LIN {X 0,Y 45.733,Z 728.488,A -85,B 0,C 180,E1 -30032.551,E2 -30032.551} C_VEL
LIN {X 0,Y 45.215,Z 723.563,A -85,B 0,C 180,E1 -30078.116,E2 -30078.116} C_VEL
LIN {X 0,Y 55.921,Z 720.857,A -85,B 0,C 180,E1 -30098.935,E2 -30098.935} C_VEL
LIN {X 0,Y 58.826,Z 720.679,A -85,B 0,C 180,E1 -30104.197,E2 -30104.197} C_VEL
LIN {X 0,Y 48.539,Z 726.04,A -85,B 0,C 180,E1 -30114.598,E2 -30114.598} C_VEL
LIN {X 0,Y 40.212,Z 730.336,A -85,B 0,C 180,E1 -30129.529,E2 -30129.529} C_VEL
LIN {X 0,Y 35.144,Z 733.679,A -85,B 0,C 180,E1 -30150.436,E2 -30150.436} C_VEL
LIN {X 0,Y 34.555,Z 735.898,A -85,B 0,C 180,E1 -30173.989,E2 -30173.989} C_VEL
LIN {X 0,Y 39.075,Z 737.272,A -85,B 0,C 180,E1 -30195.991,E2 -30195.991} C_VEL
LIN {X 0,Y 49.391,Z 737.543,A -85,B 0,C 180,E1 -30214.726,E2 -30214.726} C_VEL
LIN {X 0,Y 63.722,Z 736.291,A -85,B 0,C 180,E1 -30227.254,E2 -30227.254} C_VEL
LIN {X 0,Y 79.407,Z 733.489,A -85,B 0,C 180,E1 -30234.92,E2 -30234.92} C_VEL
LIN {X 0,Y 80.609,Z 733.2,A -85,B 0,C 180,E1 -30235.369,E2 -30235.369} C_VEL
LIN {X 0,Y 83.762,Z 732.473,A -85,B 0,C 180,E1 -30236.987,E2 -30236.987} C_VEL
LIN {X 0,Y 92.73,Z 730.259,A -85,B 0,C 180,E1 -30243.394,E2 -30243.394} C_VEL
LIN {X 0,Y 96.102,Z 729.265,A -85,B 0,C 180,E1 -30244.536,E2 -30244.536} C_VEL
LIN {X 0,Y 98.768,Z 728.439,A -85,B 0,C 180,E1 -30245.06,E2 -30245.06} C_VEL
LIN {X 0,Y 98.879,Z 728.459,A -85,B 0,C 180,E1 -30245.741,E2 -30245.741} C_VEL
LIN {X 0,Y 85.239,Z 732.788,A -85,B 0,C 180,E1 -30248.386,E2 -30248.386} C_VEL
LIN {X 0,Y 71.87,Z 736.158,A -85,B 0,C 180,E1 -30252.108,E2 -30252.108} C_VEL
LIN {X 0,Y 58.961,Z 738.548,A -85,B 0,C 180,E1 -30257.552,E2 -30257.552} C_VEL
LIN {X 0,Y 44.77,Z 740.255,A -85,B 0,C 180,E1 -30268.091,E2 -30268.091} C_VEL
LIN {X 0,Y 32.272,Z 740.603,A -85,B 0,C 180,E1 -30289.225,E2 -30289.225} C_VEL
LIN {X 0,Y 27.769,Z 739.764,A -85,B 0,C 180,E1 -30315.356,E2 -30315.356} C_VEL
LIN {X 0,Y 27.901,Z 739.026,A -85,B 0,C 180,E1 -30330.015,E2 -30330.015} C_VEL
LIN {X 0,Y 29.362,Z 736.41,A -85,B 0,C 180,E1 -30358.618,E2 -30358.618} C_VEL
LIN {X 0,Y 36.467,Z 732.693,A -85,B 0,C 180,E1 -30380.451,E2 -30380.451} C_VEL
LIN {X 0,Y 39.799,Z 730.817,A -85,B 0,C 180,E1 -30388.016,E2 -30388.016} C_VEL
LIN {X 0,Y 38.938,Z 726.095,A -85,B 0,C 180,E1 -30441.165,E2 -30441.165} C_VEL
LIN {X 0,Y 48.749,Z 723.861,A -85,B 0,C 180,E1 -30460.968,E2 -30460.968} C_VEL
LIN {X 0,Y 48.378,Z 724.351,A -85,B 0,C 180,E1 -30463.406,E2 -30463.406} C_VEL
LIN {X 0,Y 37.896,Z 729.071,A -85,B 0,C 180,E1 -30476.182,E2 -30476.182} C_VEL
LIN {X 0,Y 30.159,Z 732.784,A -85,B 0,C 180,E1 -30496.51,E2 -30496.51} C_VEL
LIN {X 0,Y 27.913,Z 734.288,A -85,B 0,C 180,E1 -30509.985,E2 -30509.985} C_VEL
LIN {X 0,Y 27.959,Z 736.485,A -85,B 0,C 180,E1 -30540.163,E2 -30540.163} C_VEL
LIN {X 0,Y 34.279,Z 737.777,A -85,B 0,C 180,E1 -30565.072,E2 -30565.072} C_VEL
LIN {X 0,Y 45.412,Z 738.013,A -85,B 0,C 180,E1 -30581.965,E2 -30581.965} C_VEL
LIN {X 0,Y 61.119,Z 736.803,A -85,B 0,C 180,E1 -30593.394,E2 -30593.394} C_VEL
LIN {X 0,Y 70.34,Z 735.461,A -85,B 0,C 180,E1 -30597.481,E2 -30597.481} C_VEL
LIN {X 0,Y 84.374,Z 732.503,A -85,B 0,C 180,E1 -30601.894,E2 -30601.894} C_VEL
LIN {X 0,Y 96.102,Z 729.265,A -85,B 0,C 180,E1 -30604.536,E2 -30604.536} C_VEL
LIN {X 0,Y 95.247,Z 729.582,A -85,B 0,C 180,E1 -30604.95,E2 -30604.95} C_VEL
LIN {X 0,Y 89.533,Z 731.374,A -85,B 0,C 180,E1 -30605.285,E2 -30605.285} C_VEL
LIN {X 0,Y 76.501,Z 734.548,A -85,B 0,C 180,E1 -30604.408,E2 -30604.408} C_VEL
LIN {X 0,Y 67.963,Z 736.139,A -85,B 0,C 180,E1 -30602.933,E2 -30602.933} C_VEL
LIN {X 0,Y 65.186,Z 736.543,A -85,B 0,C 180,E1 -30602.135,E2 -30602.135} C_VEL
LIN {X 0,Y 49.356,Z 738.175,A -85,B 0,C 180,E1 -30595.276,E2 -30595.276} C_VEL
LIN {X 0,Y 36.402,Z 738.534,A -85,B 0,C 180,E1 -30584.821,E2 -30584.821} C_VEL
LIN {X 0,Y 25.651,Z 737.78,A -85,B 0,C 180,E1 -30565.251,E2 -30565.251} C_VEL
LIN {X 0,Y 20.031,Z 736.132,A -85,B 0,C 180,E1 -30530.517,E2 -30530.517} C_VEL
LIN {X 0,Y 21.174,Z 734.546,A -85,B 0,C 180,E1 -30504.822,E2 -30504.822} C_VEL
LIN {X 0,Y 27.234,Z 731.751,A -85,B 0,C 180,E1 -30478.91,E2 -30478.91} C_VEL
LIN {X 0,Y 37.817,Z 727.643,A -85,B 0,C 180,E1 -30461.965,E2 -30461.965} C_VEL
LIN {X 0,Y 38.528,Z 727.135,A -85,B 0,C 180,E1 -30458.983,E2 -30458.983} C_VEL
LIN {X 0,Y 29.991,Z 729.275,A -85,B 0,C 180,E1 -30433.559,E2 -30433.559} C_VEL
LIN {X 0,Y 30.921,Z 731.924,A -85,B 0,C 180,E1 -30392.969,E2 -30392.969} C_VEL
LIN {X 0,Y 30.686,Z 732.637,A -85,B 0,C 180,E1 -30387.672,E2 -30387.672} C_VEL
LIN {X 0,Y 23.314,Z 735.764,A -85,B 0,C 180,E1 -30367.1,E2 -30367.1} C_VEL
LIN {X 0,Y 20.749,Z 738.425,A -85,B 0,C 180,E1 -30330.021,E2 -30330.021} C_VEL
LIN {X 0,Y 23.261,Z 739.77,A -85,B 0,C 180,E1 -30292.846,E2 -30292.846} C_VEL
LIN {X 0,Y 32.345,Z 740.149,A -85,B 0,C 180,E1 -30269.671,E2 -30269.671} C_VEL
LIN {X 0,Y 44.215,Z 739.654,A -85,B 0,C 180,E1 -30257.536,E2 -30257.536} C_VEL
LIN {X 0,Y 57.197,Z 738.196,A -85,B 0,C 180,E1 -30250.629,E2 -30250.629} C_VEL
LIN {X 0,Y 74.92,Z 734.948,A -85,B 0,C 180,E1 -30245.38,E2 -30245.38} C_VEL
LIN {X 0,Y 70.419,Z 735.773,A -85,B 0,C 180,E1 -30243.71,E2 -30243.71} C_VEL
LIN {X 0,Y 65.186,Z 736.543,A -85,B 0,C 180,E1 -30242.135,E2 -30242.135} C_VEL
LIN {X 0,Y 59.52,Z 737.347,A -85,B 0,C 180,E1 -30240.788,E2 -30240.788} C_VEL
LIN {X 0,Y 49.702,Z 738.405,A -85,B 0,C 180,E1 -30239.901,E2 -30239.901} C_VEL
LIN {X 0,Y 41.785,Z 738.909,A -85,B 0,C 180,E1 -30239.149,E2 -30239.149} C_VEL
LIN {X 0,Y 36.006,Z 738.998,A -85,B 0,C 180,E1 -30237.236,E2 -30237.236} C_VEL
LIN {X 0,Y 34.169,Z 738.96,A -85,B 0,C 180,E1 -30236.057,E2 -30236.057} C_VEL
LIN {X 0,Y 22.24,Z 738.328,A -85,B 0,C 180,E1 -30221.383,E2 -30221.383} C_VEL
LIN {X 0,Y 13.382,Z 736.754,A -85,B 0,C 180,E1 -30181.642,E2 -30181.642} C_VEL
LIN {X 0,Y 16.485,Z 734.105,A -85,B 0,C 180,E1 -30124.738,E2 -30124.738} C_VEL
LIN {X 0,Y 28.263,Z 730.197,A -85,B 0,C 180,E1 -30097.877,E2 -30097.877} C_VEL
LIN {X 0,Y 27.663,Z 730.225,A -85,B 0,C 180,E1 -30094.369,E2 -30094.369} C_VEL
LIN {X 0,Y 22.696,Z 733.126,A -85,B 0,C 180,E1 -30038.323,E2 -30038.323} C_VEL
LIN {X 0,Y 18.092,Z 735.113,A -85,B 0,C 180,E1 -30021.016,E2 -30021.016} C_VEL
LIN {X 0,Y 13.61,Z 737.823,A -85,B 0,C 180,E1 -29970.032,E2 -29970.032} C_VEL
LIN {X 0,Y 18.066,Z 739.249,A -85,B 0,C 180,E1 -29918.957,E2 -29918.957} C_VEL
LIN {X 0,Y 29.454,Z 739.669,A -85,B 0,C 180,E1 -29897.414,E2 -29897.414} C_VEL
LIN {X 0,Y 42.601,Z 739.257,A -85,B 0,C 180,E1 -29888.256,E2 -29888.256} C_VEL
LIN {X 0,Y 49.415,Z 738.654,A -85,B 0,C 180,E1 -29885.492,E2 -29885.492} C_VEL
LIN {X 0,Y 49.315,Z 738.589,A -85,B 0,C 180,E1 -29884.114,E2 -29884.114} C_VEL
LIN {X 0,Y 34.169,Z 738.96,A -85,B 0,C 180,E1 -29876.057,E2 -29876.057} C_VEL
LIN {X 0,Y 31.047,Z 738.944,A -85,B 0,C 180,E1 -29874.925,E2 -29874.925} C_VEL
LIN {X 0,Y 26.531,Z 738.96,A -85,B 0,C 180,E1 -29876.532,E2 -29876.532} C_VEL
LIN {X 0,Y 16.876,Z 738.889,A -85,B 0,C 180,E1 -29891.795,E2 -29891.795} C_VEL
LIN {X 0,Y 14.449,Z 738.697,A -85,B 0,C 180,E1 -29896.913,E2 -29896.913} C_VEL
LIN {X 0,Y 6.455,Z 737.218,A -85,B 0,C 180,E1 -29970.066,E2 -29970.066} C_VEL
LIN {X 0,Y 8.875,Z 735.956,A -85,B 0,C 180,E1 -30022.443,E2 -30022.443} C_VEL
LIN {X 0,Y 14.533,Z 734.385,A -85,B 0,C 180,E1 -30045.398,E2 -30045.398} C_VEL
LIN {X 0,Y 14.778,Z 733.855,A -85,B 0,C 180,E1 -30060.012,E2 -30060.012} C_VEL
LIN {X 0,Y 16.93,Z 733.02,A -85,B 0,C 180,E1 -30084.538,E2 -30084.538} C_VEL
LIN {X 0,Y 16.684,Z 733.156,A -85,B 0,C 180,E1 -30092.551,E2 -30092.551} C_VEL
LIN {X 0,Y 8.159,Z 735.395,A -85,B 0,C 180,E1 -30119.52,E2 -30119.52} C_VEL
LIN {X 0,Y 8.096,Z 737.341,A -85,B 0,C 180,E1 -30210.127,E2 -30210.127} C_VEL
LIN {X 0,Y 21.081,Z 738.876,A -85,B 0,C 180,E1 -30241.188,E2 -30241.188} C_VEL
LIN {X 0,Y 24.57,Z 739.141,A -85,B 0,C 180,E1 -30243.86,E2 -30243.86} C_VEL
LIN {X 0,Y 21.271,Z 739.052,A -85,B 0,C 180,E1 -30247.756,E2 -30247.756} C_VEL
LIN {X 0,Y 14.449,Z 738.697,A -85,B 0,C 180,E1 -30256.913,E2 -30256.913} C_VEL
LIN {X 0,Y 14.449,Z 738.697,A -85,B 0,C 180,E1 -30256.913,E2 -30256.913}

QRS_NEXT_CUT()

QRS_NEXT()
QRS_HOME()

END
